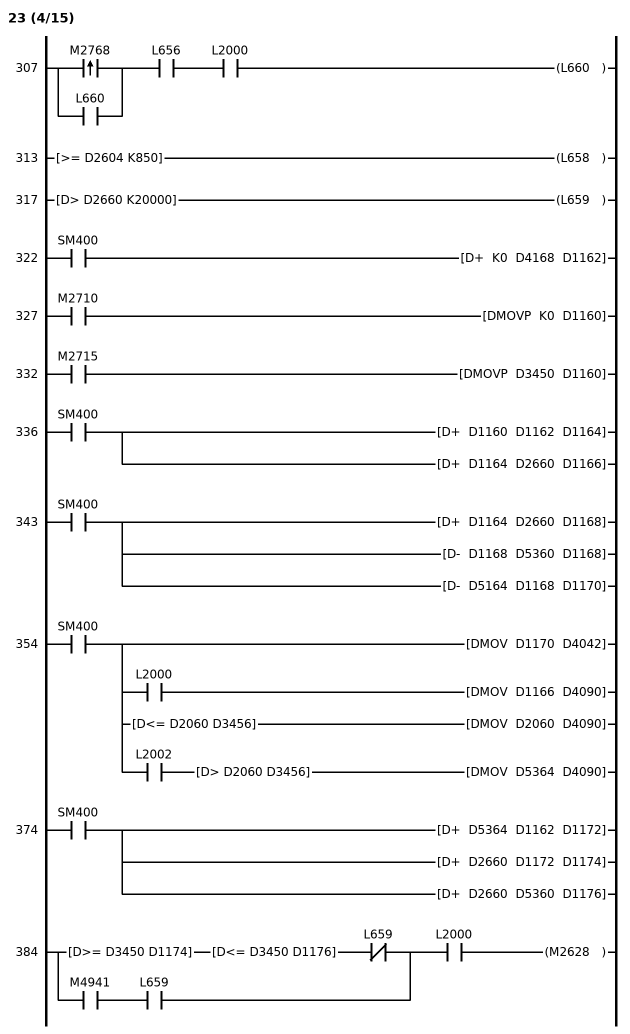
307   LDP     M2768
      OR      L660
      AND     L656
      AND     L2000
      OUT     L660
313   LD>=    D2604 K850
      OUT     L658
317   LDD>    D2660 K20000
      OUT     L659
322   LD      SM400
      D+      K0 D4168 D1162
327   LD      M2710
      DMOVP   K0 D1160
332   LD      M2715
      DMOVP   D3450 D1160
336   LD      SM400
      D+      D1160 D1162 D1164
      D+      D1164 D2660 D1166
343   LD      SM400
      D+      D1164 D2660 D1168
      D-      D1168 D5360 D1168
      D-      D5164 D1168 D1170
354   LD      SM400
      DMOV    D1170 D4042
      MPS
      AND     L2000
      DMOV    D1166 D4090
      MRD
      ANDD<=  D2060 D3456
      DMOV    D2060 D4090
      MPP
      AND     L2002
      ANDD>   D2060 D3456
      DMOV    D5364 D4090
374   LD      SM400
      D+      D5364 D1162 D1172
      D+      D2660 D1172 D1174
      D+      D2660 D5360 D1176
384   LDD>=   D3450 D1174
      ANDD<=  D3450 D1176
      ANI     L659
      LD      M4941
      AND     L659
      ORB
      AND     L2000
      OUT     M2628
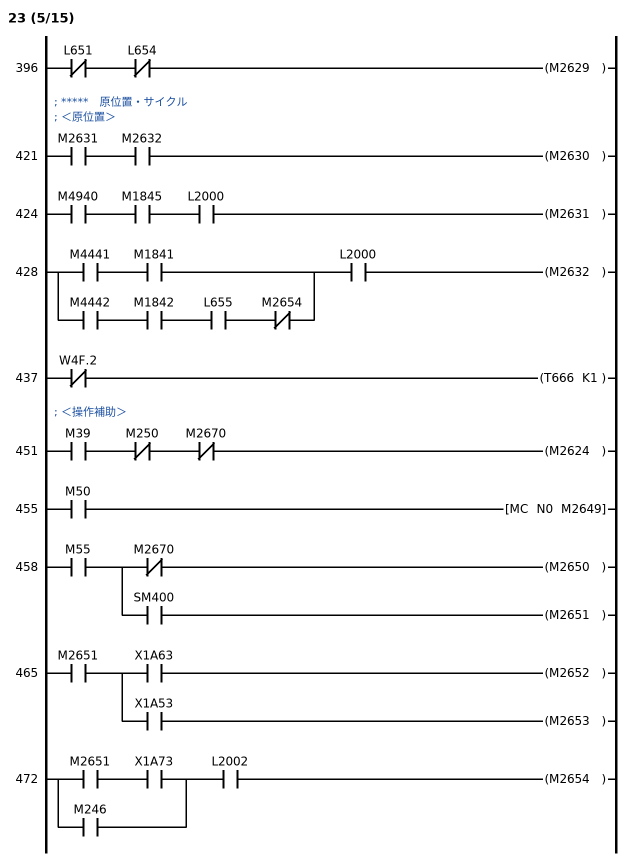
396   LDI     L651
      ANI     L654
      OUT     M2629
; *****　原位置・サイクル
; ＜原位置＞
421   LD      M2631
      AND     M2632
      OUT     M2630
424   LD      M4940
      AND     M1845
      AND     L2000
      OUT     M2631
428   LD      M4441
      AND     M1841
      LD      M4442
      AND     M1842
      AND     L655
      ANI     M2654
      ORB
      AND     L2000
      OUT     M2632
437   LDI     W4F.2
      OUT     T666 K1
; ＜操作補助＞
451   LD      M39
      ANI     M250
      ANI     M2670
      OUT     M2624
455   LD      M50
      MC      N0 M2649
458   LD      M55
      MPS
      ANI     M2670
      OUT     M2650
      MPP
      AND     SM400
      OUT     M2651
465   LD      M2651
      MPS
      AND     X1A63
      OUT     M2652
      MPP
      AND     X1A53
      OUT     M2653
472   LD      M2651
      AND     X1A73
      OR      M246
      AND     L2002
      OUT     M2654
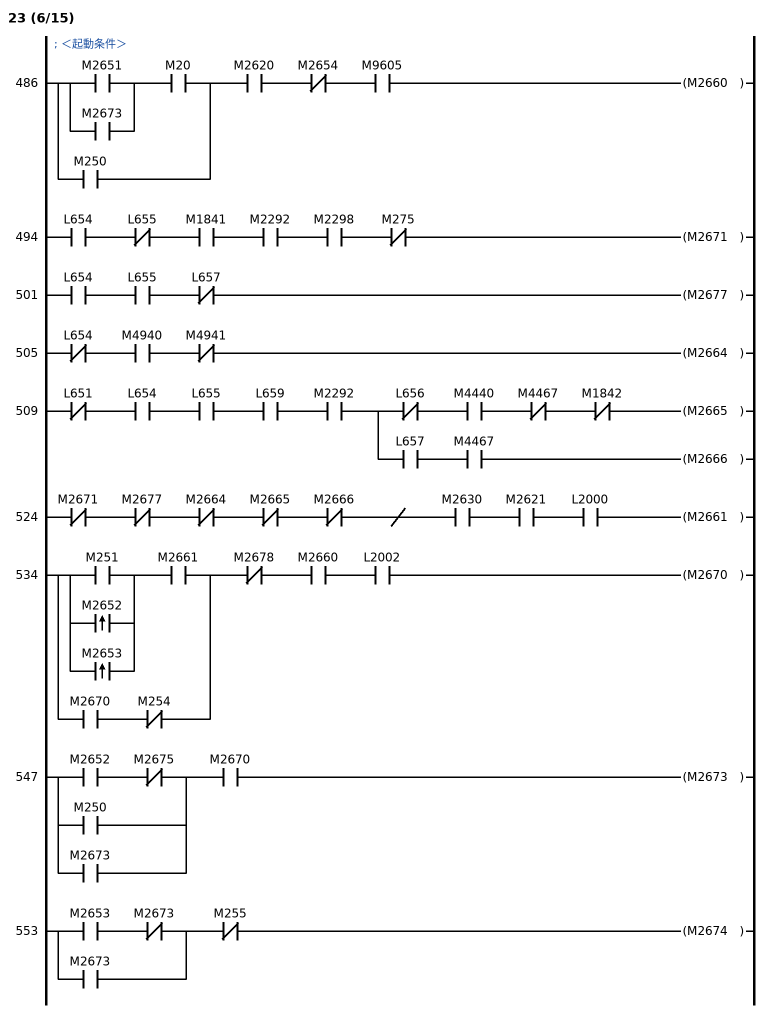
; ＜起動条件＞
486   LD      M2651
      OR      M2673
      AND     M20
      OR      M250
      AND     M2620
      ANI     M2654
      AND     M9605
      OUT     M2660
494   LD      L654
      ANI     L655
      AND     M1841
      AND     M2292
      AND     M2298
      ANI     M275
      OUT     M2671
501   LD      L654
      AND     L655
      ANI     L657
      OUT     M2677
505   LDI     L654
      AND     M4940
      ANI     M4941
      OUT     M2664
509   LDI     L651
      AND     L654
      AND     L655
      AND     L659
      AND     M2292
      MPS
      ANI     L656
      AND     M4440
      ANI     M4467
      ANI     M1842
      OUT     M2665
      MPP
      AND     L657
      AND     M4467
      OUT     M2666
524   LDI     M2671
      ANI     M2677
      ANI     M2664
      ANI     M2665
      ANI     M2666
      INV
      AND     M2630
      AND     M2621
      AND     L2000
      OUT     M2661
534   LD      M251
      ORP     M2652
      ORP     M2653
      AND     M2661
      LD      M2670
      ANI     M254
      ORB
      ANI     M2678
      AND     M2660
      AND     L2002
      OUT     M2670
547   LD      M2652
      ANI     M2675
      OR      M250
      OR      M2673
      AND     M2670
      OUT     M2673
553   LD      M2653
      ANI     M2673
      OR      M2673
      ANI     M255
      OUT     M2674
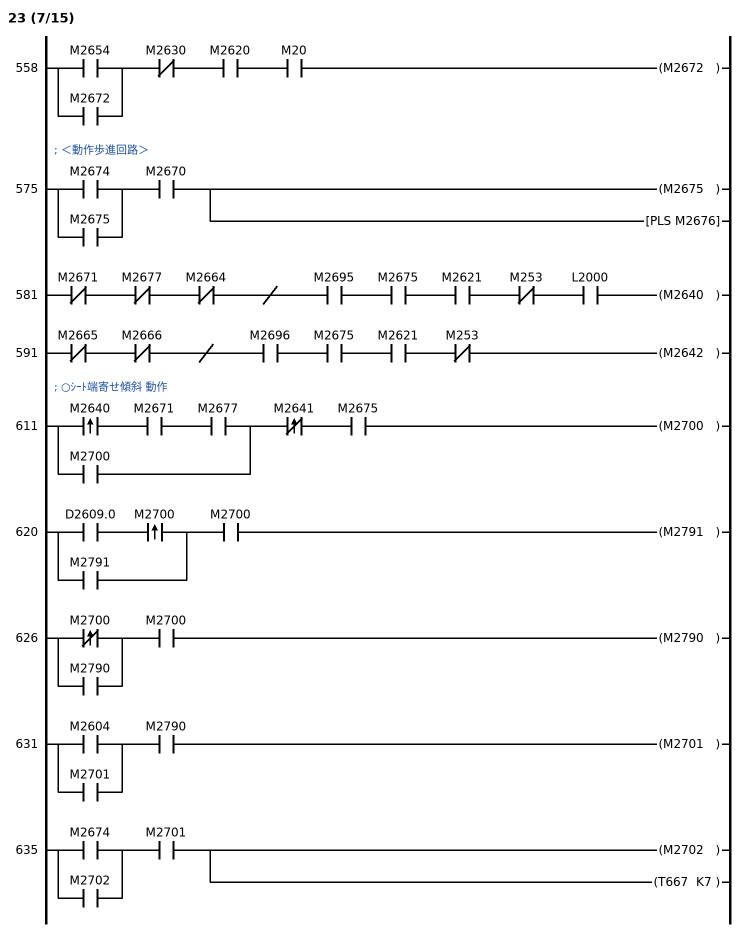
558   LD      M2654
      OR      M2672
      ANI     M2630
      AND     M2620
      AND     M20
      OUT     M2672
; ＜動作歩進回路＞
575   LD      M2674
      OR      M2675
      AND     M2670
      OUT     M2675
      PLS     M2676
581   LDI     M2671
      ANI     M2677
      ANI     M2664
      INV
      AND     M2695
      AND     M2675
      AND     M2621
      ANI     M253
      AND     L2000
      OUT     M2640
591   LDI     M2665
      ANI     M2666
      INV
      AND     M2696
      AND     M2675
      AND     M2621
      ANI     M253
      OUT     M2642
; ○ｼｰﾄ端寄せ傾斜 動作
611   LDP     M2640
      AND     M2671
      AND     M2677
      OR      M2700
      ANDPI   M2641
      AND     M2675
      OUT     M2700
620   LD      D2609.0
      ANDP    M2700
      OR      M2791
      AND     M2700
      OUT     M2791
626   LDPI    M2700
      OR      M2790
      AND     M2700
      OUT     M2790
631   LD      M2604
      OR      M2701
      AND     M2790
      OUT     M2701
635   LD      M2674
      OR      M2702
      AND     M2701
      OUT     M2702
      OUT     T667 K7
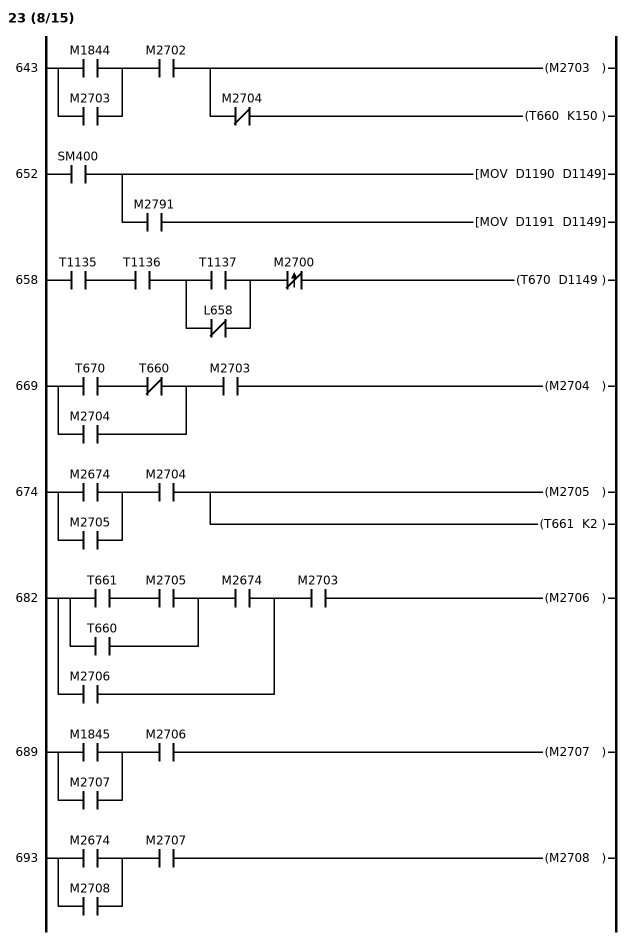
643   LD      M1844
      OR      M2703
      AND     M2702
      OUT     M2703
      ANI     M2704
      OUT     T660 K150
652   LD      SM400
      MOV     D1190 D1149
      AND     M2791
      MOV     D1191 D1149
658   LD      T1135
      AND     T1136
      LD      T1137
      ORI     L658
      ANB
      ANDPI   M2700
      OUT     T670 D1149
669   LD      T670
      ANI     T660
      OR      M2704
      AND     M2703
      OUT     M2704
674   LD      M2674
      OR      M2705
      AND     M2704
      OUT     M2705
      OUT     T661 K2
682   LD      T661
      AND     M2705
      OR      T660
      AND     M2674
      OR      M2706
      AND     M2703
      OUT     M2706
689   LD      M1845
      OR      M2707
      AND     M2706
      OUT     M2707
693   LD      M2674
      OR      M2708
      AND     M2707
      OUT     M2708
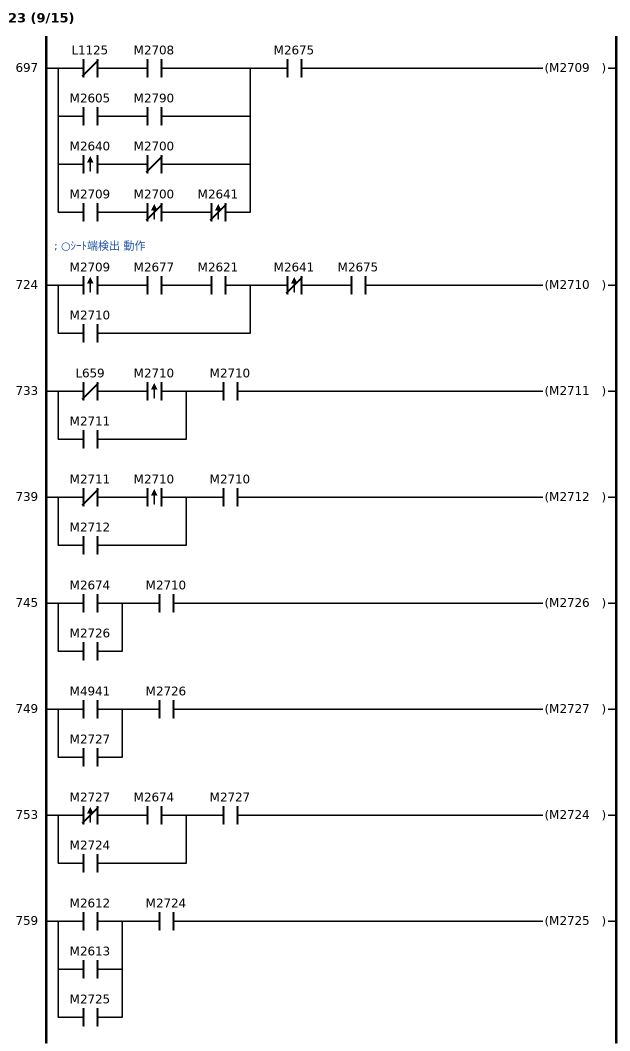
697   LDI     L1125
      AND     M2708
      LD      M2605
      AND     M2790
      ORB
      LDP     M2640
      ANI     M2700
      ORB
      LD      M2709
      ANDPI   M2700
      ANDPI   M2641
      ORB
      AND     M2675
      OUT     M2709
; ○ｼｰﾄ端検出 動作
724   LDP     M2709
      AND     M2677
      AND     M2621
      OR      M2710
      ANDPI   M2641
      AND     M2675
      OUT     M2710
733   LDI     L659
      ANDP    M2710
      OR      M2711
      AND     M2710
      OUT     M2711
739   LDI     M2711
      ANDP    M2710
      OR      M2712
      AND     M2710
      OUT     M2712
745   LD      M2674
      OR      M2726
      AND     M2710
      OUT     M2726
749   LD      M4941
      OR      M2727
      AND     M2726
      OUT     M2727
753   LDPI    M2727
      AND     M2674
      OR      M2724
      AND     M2727
      OUT     M2724
759   LD      M2612
      OR      M2613
      OR      M2725
      AND     M2724
      OUT     M2725
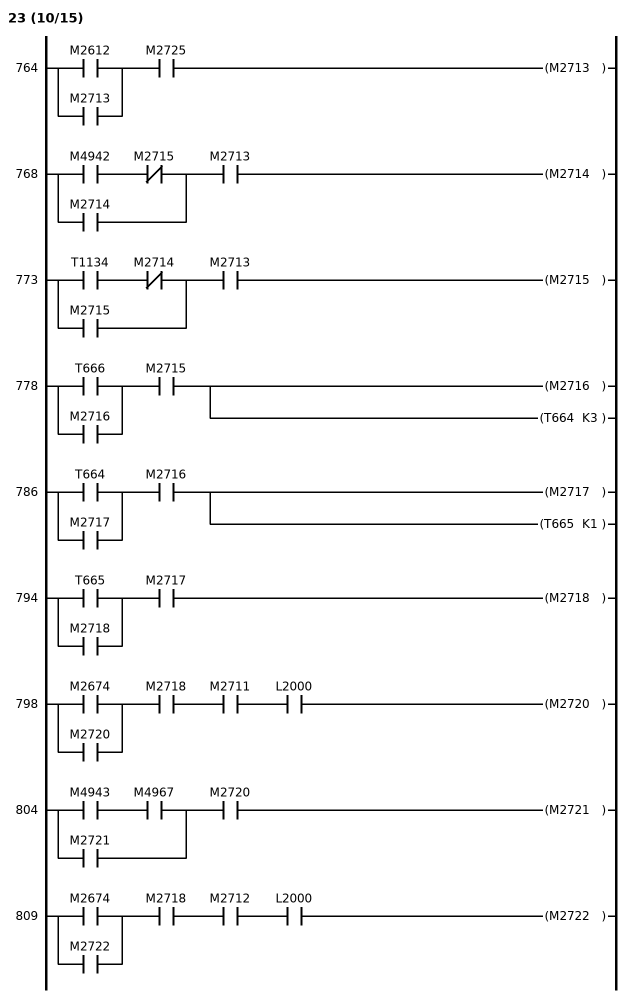
764   LD      M2612
      OR      M2713
      AND     M2725
      OUT     M2713
768   LD      M4942
      ANI     M2715
      OR      M2714
      AND     M2713
      OUT     M2714
773   LD      T1134
      ANI     M2714
      OR      M2715
      AND     M2713
      OUT     M2715
778   LD      T666
      OR      M2716
      AND     M2715
      OUT     M2716
      OUT     T664 K3
786   LD      T664
      OR      M2717
      AND     M2716
      OUT     M2717
      OUT     T665 K1
794   LD      T665
      OR      M2718
      AND     M2717
      OUT     M2718
798   LD      M2674
      OR      M2720
      AND     M2718
      AND     M2711
      AND     L2000
      OUT     M2720
804   LD      M4943
      AND     M4967
      OR      M2721
      AND     M2720
      OUT     M2721
809   LD      M2674
      OR      M2722
      AND     M2718
      AND     M2712
      AND     L2000
      OUT     M2722
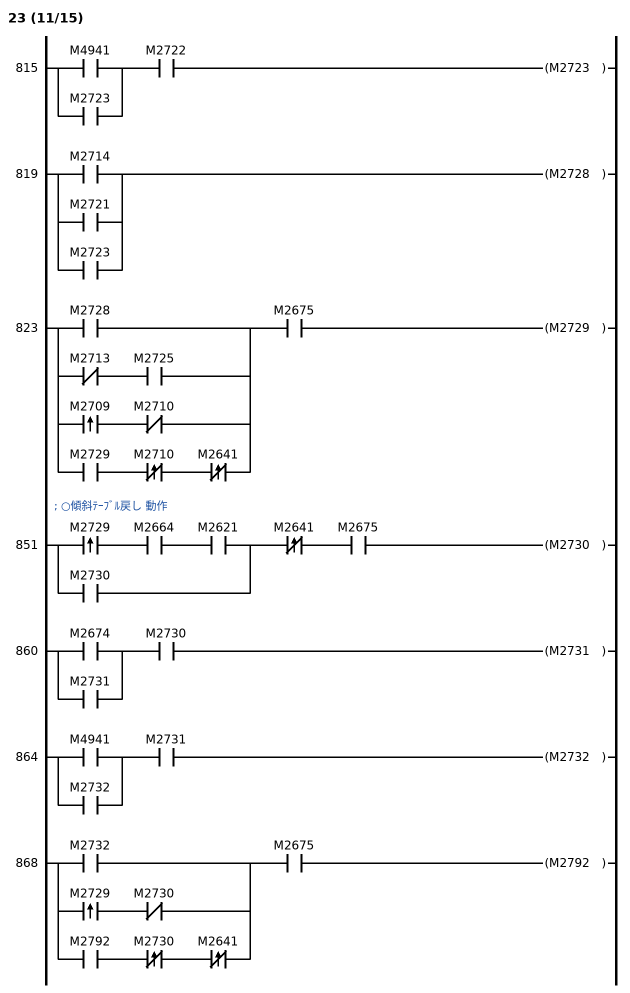
815   LD      M4941
      OR      M2723
      AND     M2722
      OUT     M2723
819   LD      M2714
      OR      M2721
      OR      M2723
      OUT     M2728
823   LD      M2728
      LDI     M2713
      AND     M2725
      ORB
      LDP     M2709
      ANI     M2710
      ORB
      LD      M2729
      ANDPI   M2710
      ANDPI   M2641
      ORB
      AND     M2675
      OUT     M2729
; ○傾斜ﾃｰﾌﾞﾙ戻し 動作
851   LDP     M2729
      AND     M2664
      AND     M2621
      OR      M2730
      ANDPI   M2641
      AND     M2675
      OUT     M2730
860   LD      M2674
      OR      M2731
      AND     M2730
      OUT     M2731
864   LD      M4941
      OR      M2732
      AND     M2731
      OUT     M2732
868   LD      M2732
      LDP     M2729
      ANI     M2730
      ORB
      LD      M2792
      ANDPI   M2730
      ANDPI   M2641
      ORB
      AND     M2675
      OUT     M2792
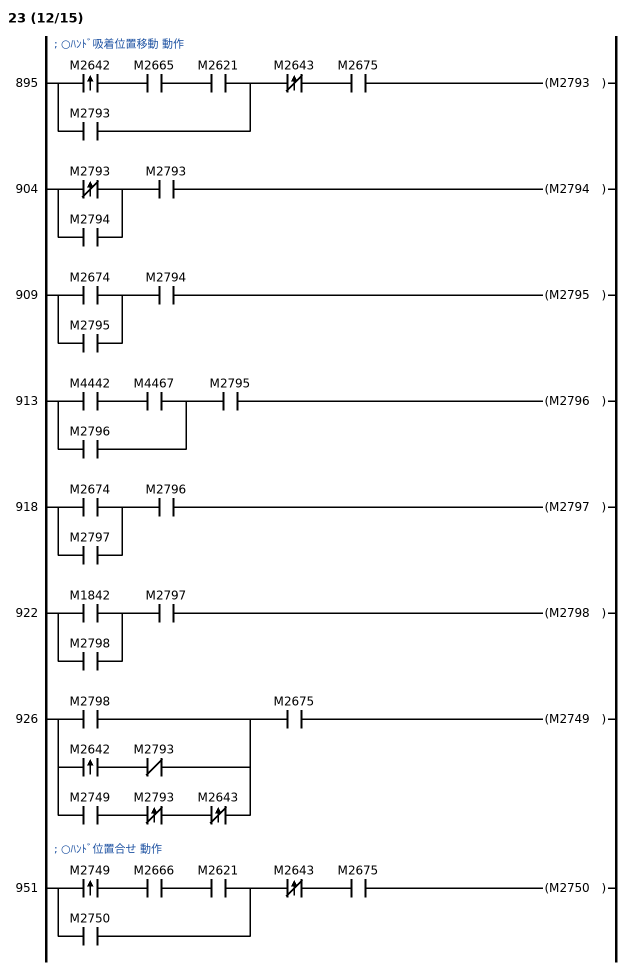
; ○ﾊﾝﾄﾞ吸着位置移動 動作
895   LDP     M2642
      AND     M2665
      AND     M2621
      OR      M2793
      ANDPI   M2643
      AND     M2675
      OUT     M2793
904   LDPI    M2793
      OR      M2794
      AND     M2793
      OUT     M2794
909   LD      M2674
      OR      M2795
      AND     M2794
      OUT     M2795
913   LD      M4442
      AND     M4467
      OR      M2796
      AND     M2795
      OUT     M2796
918   LD      M2674
      OR      M2797
      AND     M2796
      OUT     M2797
922   LD      M1842
      OR      M2798
      AND     M2797
      OUT     M2798
926   LD      M2798
      LDP     M2642
      ANI     M2793
      ORB
      LD      M2749
      ANDPI   M2793
      ANDPI   M2643
      ORB
      AND     M2675
      OUT     M2749
; ○ﾊﾝﾄﾞ位置合せ 動作
951   LDP     M2749
      AND     M2666
      AND     M2621
      OR      M2750
      ANDPI   M2643
      AND     M2675
      OUT     M2750
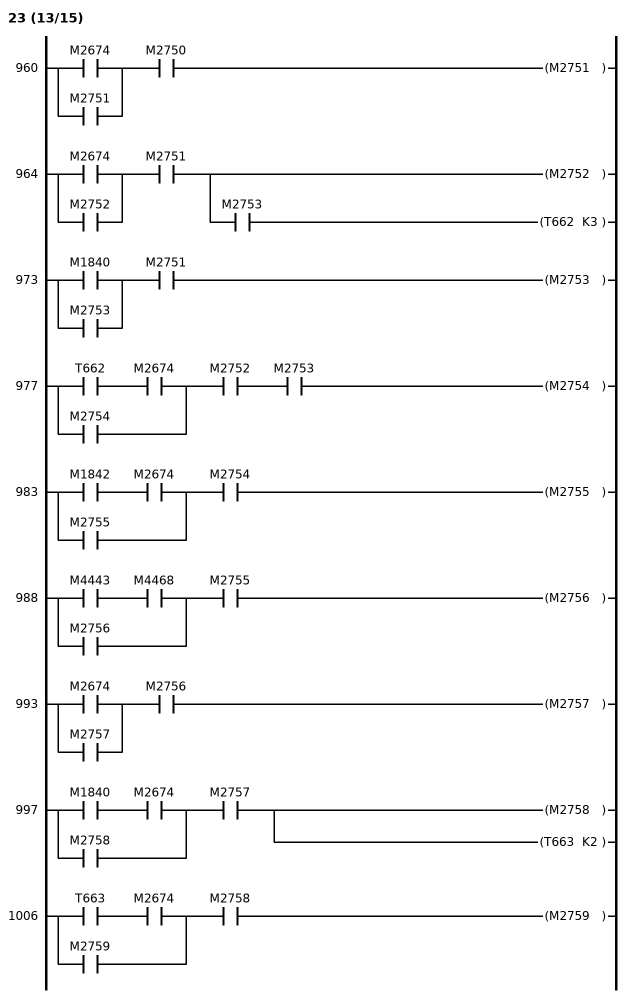
960   LD      M2674
      OR      M2751
      AND     M2750
      OUT     M2751
964   LD      M2674
      OR      M2752
      AND     M2751
      OUT     M2752
      AND     M2753
      OUT     T662 K3
973   LD      M1840
      OR      M2753
      AND     M2751
      OUT     M2753
977   LD      T662
      AND     M2674
      OR      M2754
      AND     M2752
      AND     M2753
      OUT     M2754
983   LD      M1842
      AND     M2674
      OR      M2755
      AND     M2754
      OUT     M2755
988   LD      M4443
      AND     M4468
      OR      M2756
      AND     M2755
      OUT     M2756
993   LD      M2674
      OR      M2757
      AND     M2756
      OUT     M2757
997   LD      M1840
      AND     M2674
      OR      M2758
      AND     M2757
      OUT     M2758
      OUT     T663 K2
1006  LD      T663
      AND     M2674
      OR      M2759
      AND     M2758
      OUT     M2759
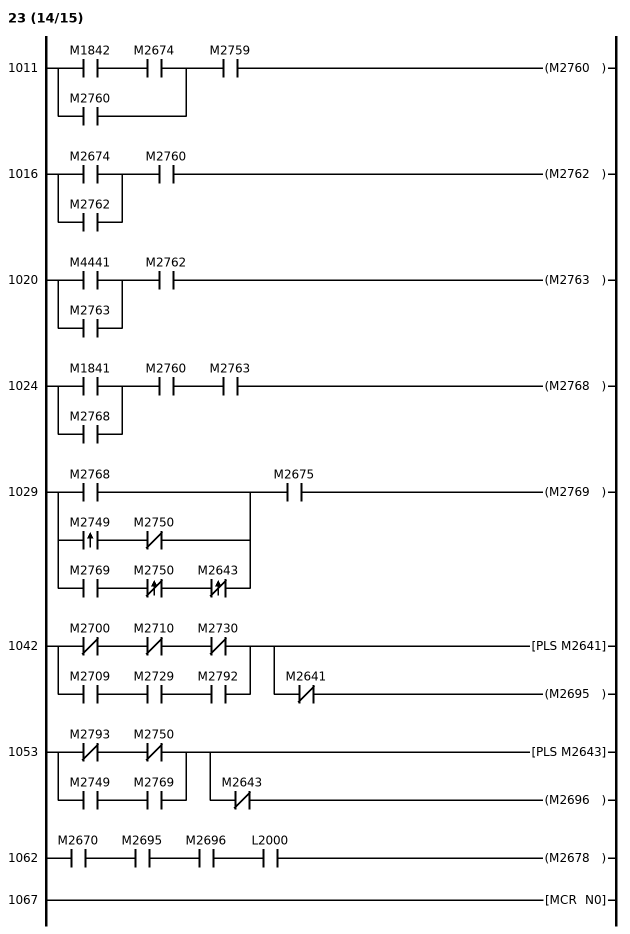
1011  LD      M1842
      AND     M2674
      OR      M2760
      AND     M2759
      OUT     M2760
1016  LD      M2674
      OR      M2762
      AND     M2760
      OUT     M2762
1020  LD      M4441
      OR      M2763
      AND     M2762
      OUT     M2763
1024  LD      M1841
      OR      M2768
      AND     M2760
      AND     M2763
      OUT     M2768
1029  LD      M2768
      LDP     M2749
      ANI     M2750
      ORB
      LD      M2769
      ANDPI   M2750
      ANDPI   M2643
      ORB
      AND     M2675
      OUT     M2769
1042  LDI     M2700
      ANI     M2710
      ANI     M2730
      LD      M2709
      AND     M2729
      AND     M2792
      ORB
      PLS     M2641
      ANI     M2641
      OUT     M2695
1053  LDI     M2793
      ANI     M2750
      LD      M2749
      AND     M2769
      ORB
      PLS     M2643
      ANI     M2643
      OUT     M2696
1062  LD      M2670
      AND     M2695
      AND     M2696
      AND     L2000
      OUT     M2678
1067  MCR     N0
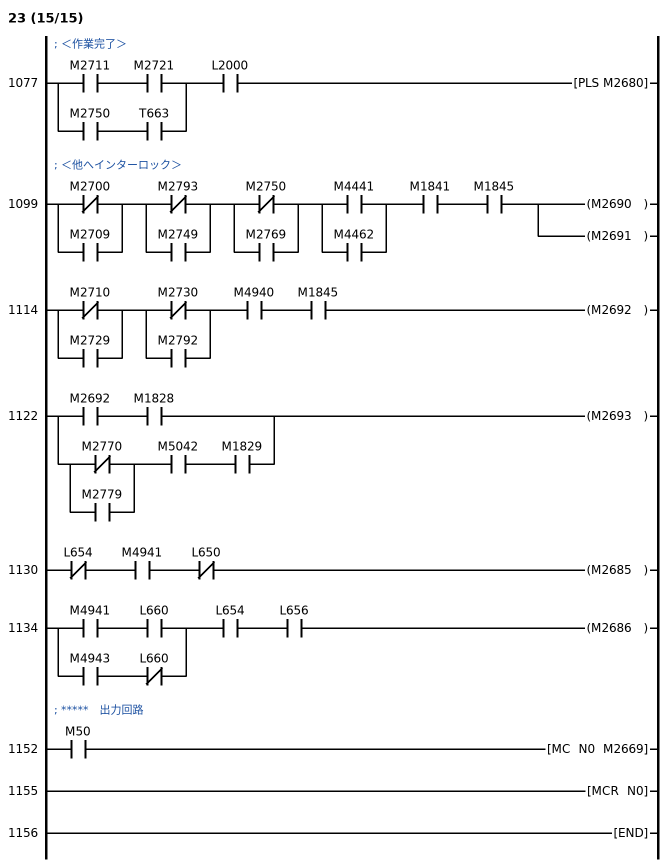
; ＜作業完了＞
1077  LD      M2711
      AND     M2721
      LD      M2750
      AND     T663
      ORB
      AND     L2000
      PLS     M2680
; ＜他へインターロック＞
1099  LDI     M2700
      OR      M2709
      LDI     M2793
      OR      M2749
      ANB
      LDI     M2750
      OR      M2769
      ANB
      LD      M4441
      OR      M4462
      ANB
      AND     M1841
      AND     M1845
      OUT     M2690
      OUT     M2691
1114  LDI     M2710
      OR      M2729
      LDI     M2730
      OR      M2792
      ANB
      AND     M4940
      AND     M1845
      OUT     M2692
1122  LD      M2692
      AND     M1828
      LDI     M2770
      OR      M2779
      AND     M5042
      AND     M1829
      ORB
      OUT     M2693
1130  LDI     L654
      AND     M4941
      ANI     L650
      OUT     M2685
1134  LD      M4941
      AND     L660
      LD      M4943
      ANI     L660
      ORB
      AND     L654
      AND     L656
      OUT     M2686
; *****　出力回路
1152  LD      M50
      MC      N0 M2669
1155  MCR     N0
1156  END
END_PROGRAM

PROGRAM 24
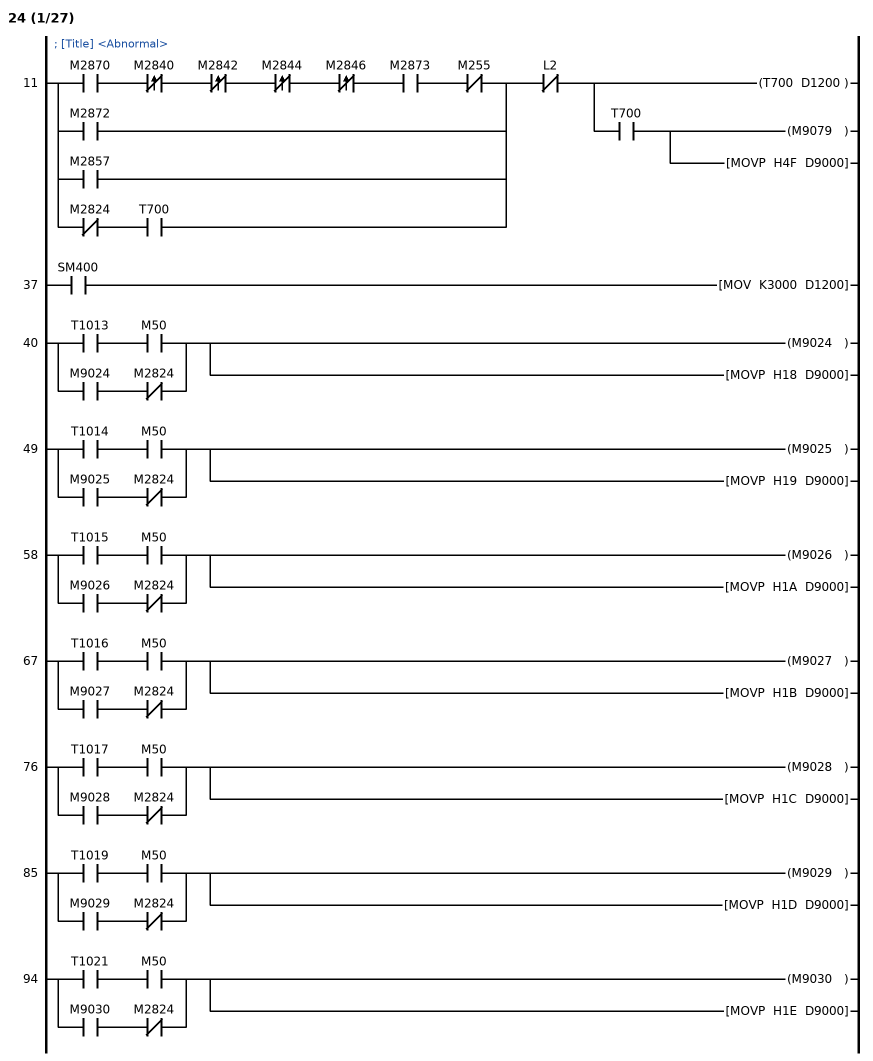
; [Title] <Abnormal>
11    LD      M2870
      ANDPI   M2840
      ANDPI   M2842
      ANDPI   M2844
      ANDPI   M2846
      AND     M2873
      ANI     M255
      OR      M2872
      OR      M2857
      LDI     M2824
      AND     T700
      ORB
      ANI     L2
      OUT     T700 D1200
      AND     T700
      OUT     M9079
      MOVP    H4F D9000
37    LD      SM400
      MOV     K3000 D1200
40    LD      T1013
      AND     M50
      LD      M9024
      ANI     M2824
      ORB
      OUT     M9024
      MOVP    H18 D9000
49    LD      T1014
      AND     M50
      LD      M9025
      ANI     M2824
      ORB
      OUT     M9025
      MOVP    H19 D9000
58    LD      T1015
      AND     M50
      LD      M9026
      ANI     M2824
      ORB
      OUT     M9026
      MOVP    H1A D9000
67    LD      T1016
      AND     M50
      LD      M9027
      ANI     M2824
      ORB
      OUT     M9027
      MOVP    H1B D9000
76    LD      T1017
      AND     M50
      LD      M9028
      ANI     M2824
      ORB
      OUT     M9028
      MOVP    H1C D9000
85    LD      T1019
      AND     M50
      LD      M9029
      ANI     M2824
      ORB
      OUT     M9029
      MOVP    H1D D9000
94    LD      T1021
      AND     M50
      LD      M9030
      ANI     M2824
      ORB
      OUT     M9030
      MOVP    H1E D9000
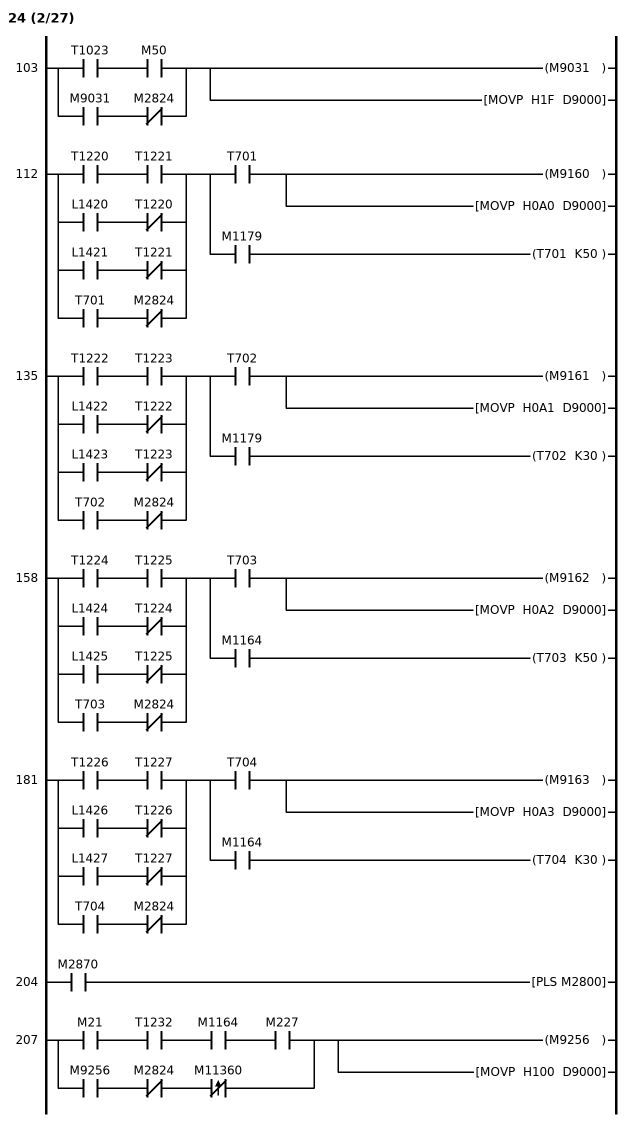
103   LD      T1023
      AND     M50
      LD      M9031
      ANI     M2824
      ORB
      OUT     M9031
      MOVP    H1F D9000
112   LD      T1220
      AND     T1221
      LD      L1420
      ANI     T1220
      ORB
      LD      L1421
      ANI     T1221
      ORB
      LD      T701
      ANI     M2824
      ORB
      MPS
      AND     T701
      OUT     M9160
      MOVP    H0A0 D9000
      MPP
      AND     M1179
      OUT     T701 K50
135   LD      T1222
      AND     T1223
      LD      L1422
      ANI     T1222
      ORB
      LD      L1423
      ANI     T1223
      ORB
      LD      T702
      ANI     M2824
      ORB
      MPS
      AND     T702
      OUT     M9161
      MOVP    H0A1 D9000
      MPP
      AND     M1179
      OUT     T702 K30
158   LD      T1224
      AND     T1225
      LD      L1424
      ANI     T1224
      ORB
      LD      L1425
      ANI     T1225
      ORB
      LD      T703
      ANI     M2824
      ORB
      MPS
      AND     T703
      OUT     M9162
      MOVP    H0A2 D9000
      MPP
      AND     M1164
      OUT     T703 K50
181   LD      T1226
      AND     T1227
      LD      L1426
      ANI     T1226
      ORB
      LD      L1427
      ANI     T1227
      ORB
      LD      T704
      ANI     M2824
      ORB
      MPS
      AND     T704
      OUT     M9163
      MOVP    H0A3 D9000
      MPP
      AND     M1164
      OUT     T704 K30
204   LD      M2870
      PLS     M2800
207   LD      M21
      AND     T1232
      AND     M1164
      AND     M227
      LD      M9256
      ANI     M2824
      ANDPI   M11360
      ORB
      OUT     M9256
      MOVP    H100 D9000
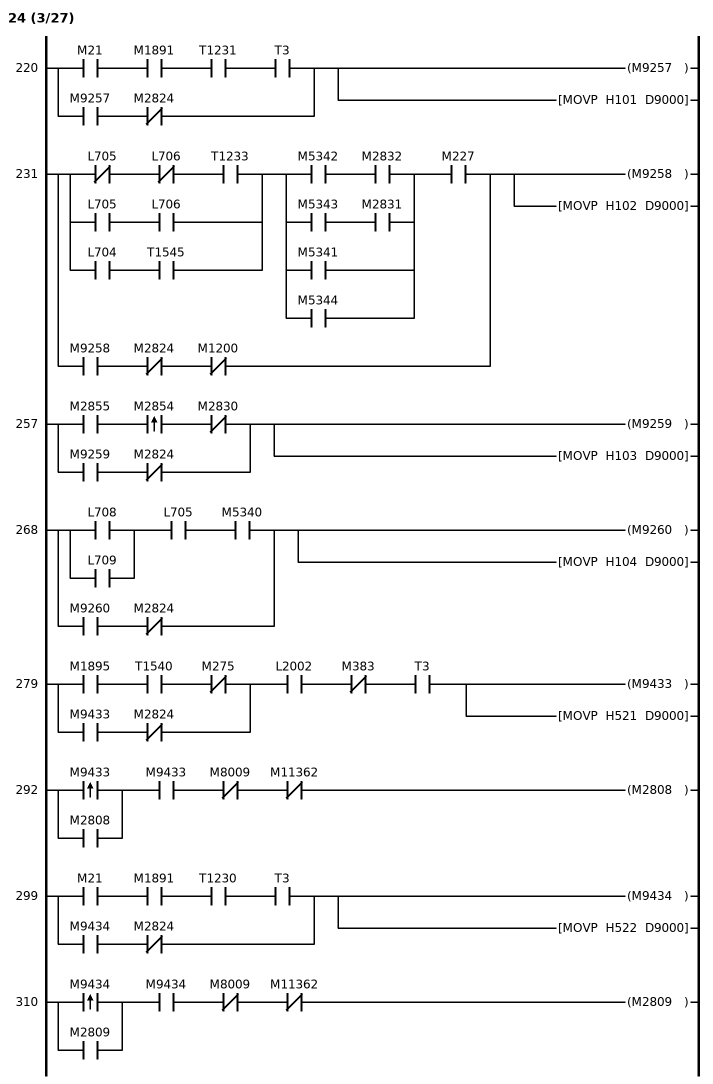
220   LD      M21
      AND     M1891
      AND     T1231
      AND     T3
      LD      M9257
      ANI     M2824
      ORB
      OUT     M9257
      MOVP    H101 D9000
231   LDI     L705
      ANI     L706
      AND     T1233
      LD      L705
      AND     L706
      ORB
      LD      L704
      AND     T1545
      ORB
      LD      M5342
      AND     M2832
      LD      M5343
      AND     M2831
      ORB
      OR      M5341
      OR      M5344
      ANB
      AND     M227
      LD      M9258
      ANI     M2824
      ANI     M1200
      ORB
      OUT     M9258
      MOVP    H102 D9000
257   LD      M2855
      ANDP    M2854
      ANI     M2830
      LD      M9259
      ANI     M2824
      ORB
      OUT     M9259
      MOVP    H103 D9000
268   LD      L708
      OR      L709
      AND     L705
      AND     M5340
      LD      M9260
      ANI     M2824
      ORB
      OUT     M9260
      MOVP    H104 D9000
279   LD      M1895
      AND     T1540
      ANI     M275
      LD      M9433
      ANI     M2824
      ORB
      AND     L2002
      ANI     M383
      AND     T3
      OUT     M9433
      MOVP    H521 D9000
292   LDP     M9433
      OR      M2808
      AND     M9433
      ANI     M8009
      ANI     M11362
      OUT     M2808
299   LD      M21
      AND     M1891
      AND     T1230
      AND     T3
      LD      M9434
      ANI     M2824
      ORB
      OUT     M9434
      MOVP    H522 D9000
310   LDP     M9434
      OR      M2809
      AND     M9434
      ANI     M8009
      ANI     M11362
      OUT     M2809
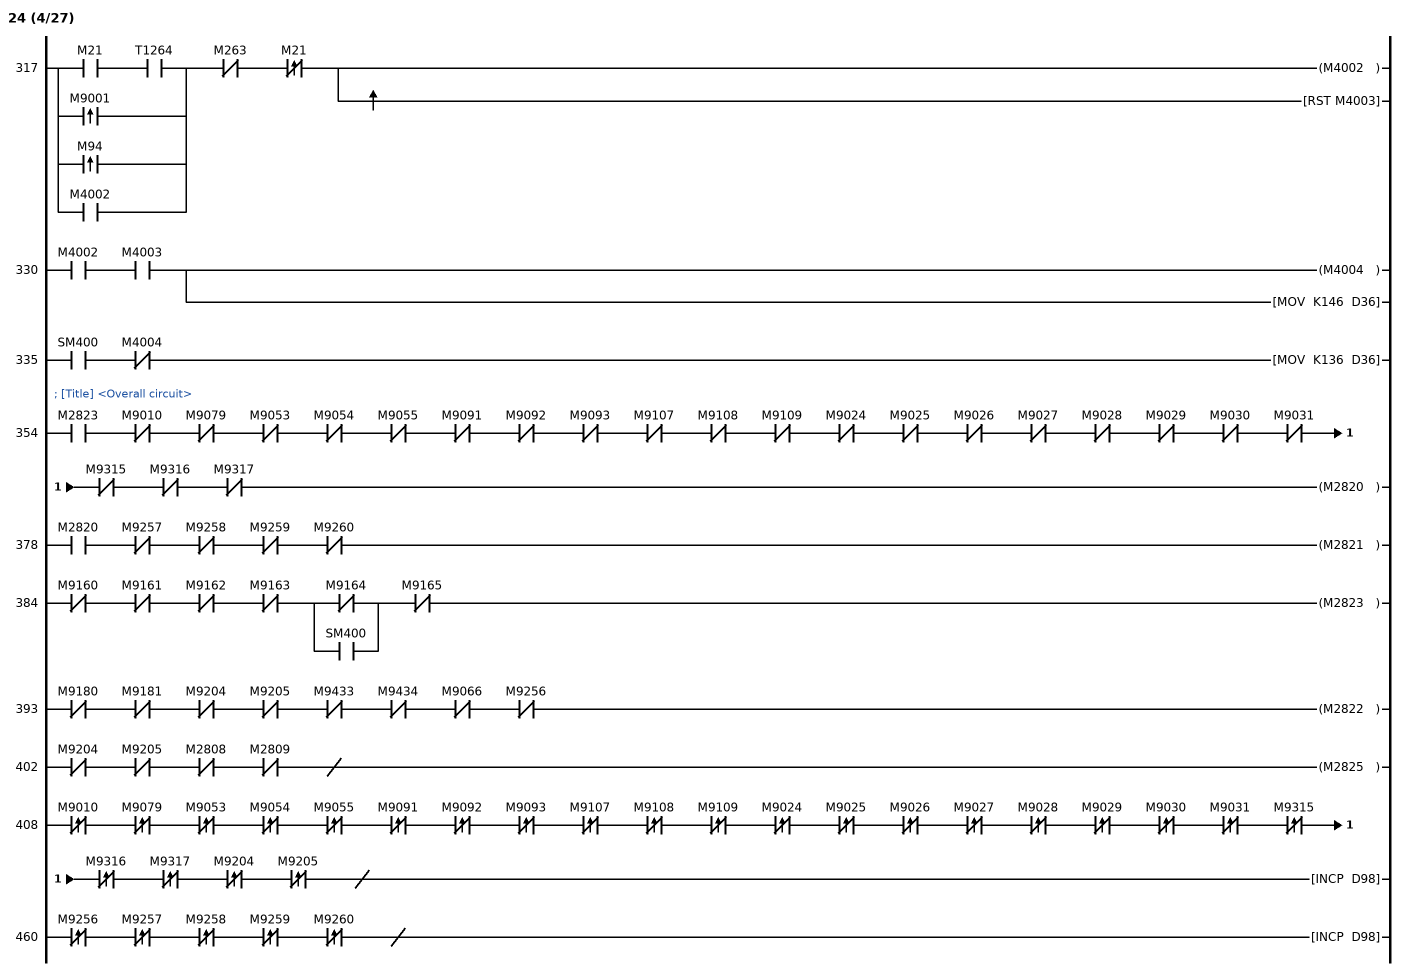
317   LD      M21
      AND     T1264
      ORP     M9001
      ORP     M94
      OR      M4002
      ANI     M263
      ANDPI   M21
      OUT     M4002
      MEP
      RST     M4003
330   LD      M4002
      AND     M4003
      OUT     M4004
      MOV     K146 D36
335   LD      SM400
      ANI     M4004
      MOV     K136 D36
; [Title] <Overall circuit>
354   LD      M2823
      ANI     M9010
      ANI     M9079
      ANI     M9053
      ANI     M9054
      ANI     M9055
      ANI     M9091
      ANI     M9092
      ANI     M9093
      ANI     M9107
      ANI     M9108
      ANI     M9109
      ANI     M9024
      ANI     M9025
      ANI     M9026
      ANI     M9027
      ANI     M9028
      ANI     M9029
      ANI     M9030
      ANI     M9031
      ANI     M9315
      ANI     M9316
      ANI     M9317
      OUT     M2820
378   LD      M2820
      ANI     M9257
      ANI     M9258
      ANI     M9259
      ANI     M9260
      OUT     M2821
384   LDI     M9160
      ANI     M9161
      ANI     M9162
      ANI     M9163
      LDI     M9164
      OR      SM400
      ANB
      ANI     M9165
      OUT     M2823
393   LDI     M9180
      ANI     M9181
      ANI     M9204
      ANI     M9205
      ANI     M9433
      ANI     M9434
      ANI     M9066
      ANI     M9256
      OUT     M2822
402   LDI     M9204
      ANI     M9205
      ANI     M2808
      ANI     M2809
      INV
      OUT     M2825
408   LDPI    M9010
      ANDPI   M9079
      ANDPI   M9053
      ANDPI   M9054
      ANDPI   M9055
      ANDPI   M9091
      ANDPI   M9092
      ANDPI   M9093
      ANDPI   M9107
      ANDPI   M9108
      ANDPI   M9109
      ANDPI   M9024
      ANDPI   M9025
      ANDPI   M9026
      ANDPI   M9027
      ANDPI   M9028
      ANDPI   M9029
      ANDPI   M9030
      ANDPI   M9031
      ANDPI   M9315
      ANDPI   M9316
      ANDPI   M9317
      ANDPI   M9204
      ANDPI   M9205
      INV
      INCP    D98
460   LDPI    M9256
      ANDPI   M9257
      ANDPI   M9258
      ANDPI   M9259
      ANDPI   M9260
      INV
      INCP    D98
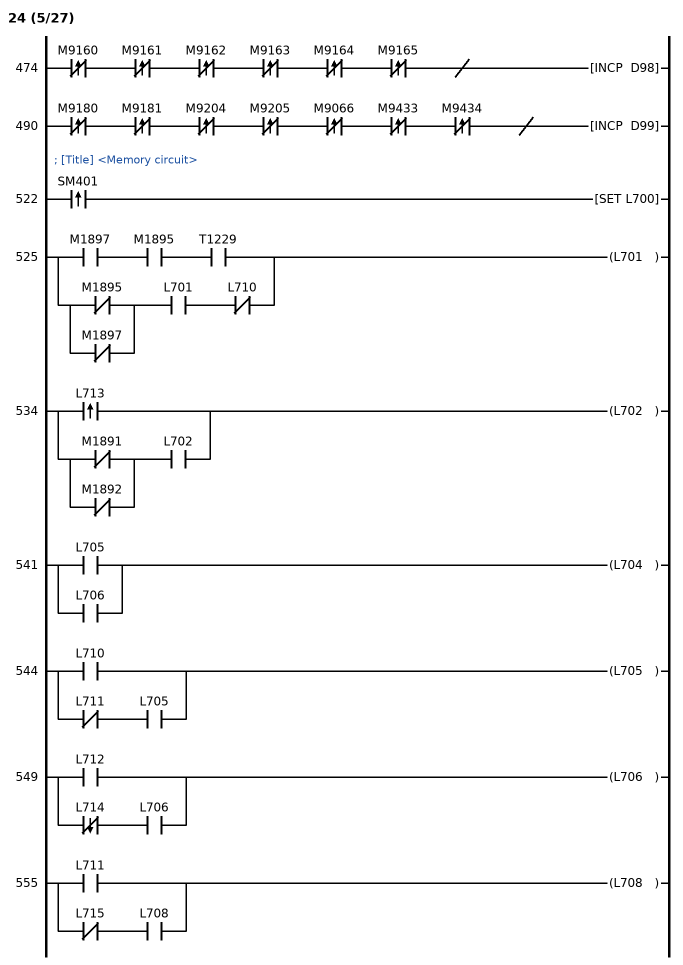
474   LDPI    M9160
      ANDPI   M9161
      ANDPI   M9162
      ANDPI   M9163
      ANDPI   M9164
      ANDPI   M9165
      INV
      INCP    D98
490   LDPI    M9180
      ANDPI   M9181
      ANDPI   M9204
      ANDPI   M9205
      ANDPI   M9066
      ANDPI   M9433
      ANDPI   M9434
      INV
      INCP    D99
; [Title] <Memory circuit>
522   LDP     SM401
      SET     L700
525   LD      M1897
      AND     M1895
      AND     T1229
      LDI     M1895
      ORI     M1897
      AND     L701
      ANI     L710
      ORB
      OUT     L701
534   LDP     L713
      LDI     M1891
      ORI     M1892
      AND     L702
      ORB
      OUT     L702
541   LD      L705
      OR      L706
      OUT     L704
544   LD      L710
      LDI     L711
      AND     L705
      ORB
      OUT     L705
549   LD      L712
      LDFI    L714
      AND     L706
      ORB
      OUT     L706
555   LD      L711
      LDI     L715
      AND     L708
      ORB
      OUT     L708
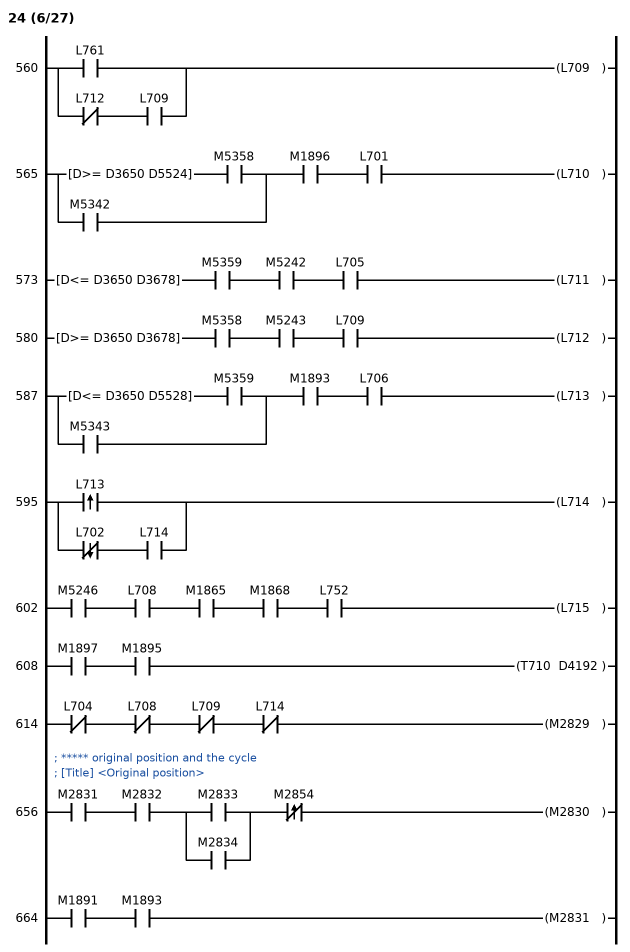
560   LD      L761
      LDI     L712
      AND     L709
      ORB
      OUT     L709
565   LDD>=   D3650 D5524
      AND     M5358
      OR      M5342
      AND     M1896
      AND     L701
      OUT     L710
573   LDD<=   D3650 D3678
      AND     M5359
      AND     M5242
      AND     L705
      OUT     L711
580   LDD>=   D3650 D3678
      AND     M5358
      AND     M5243
      AND     L709
      OUT     L712
587   LDD<=   D3650 D5528
      AND     M5359
      OR      M5343
      AND     M1893
      AND     L706
      OUT     L713
595   LDP     L713
      LDFI    L702
      AND     L714
      ORB
      OUT     L714
602   LD      M5246
      AND     L708
      AND     M1865
      AND     M1868
      AND     L752
      OUT     L715
608   LD      M1897
      AND     M1895
      OUT     T710 D4192
614   LDI     L704
      ANI     L708
      ANI     L709
      ANI     L714
      OUT     M2829
; ***** original position and the cycle
; [Title] <Original position>
656   LD      M2831
      AND     M2832
      LD      M2833
      OR      M2834
      ANB
      ANDPI   M2854
      OUT     M2830
664   LD      M1891
      AND     M1893
      OUT     M2831
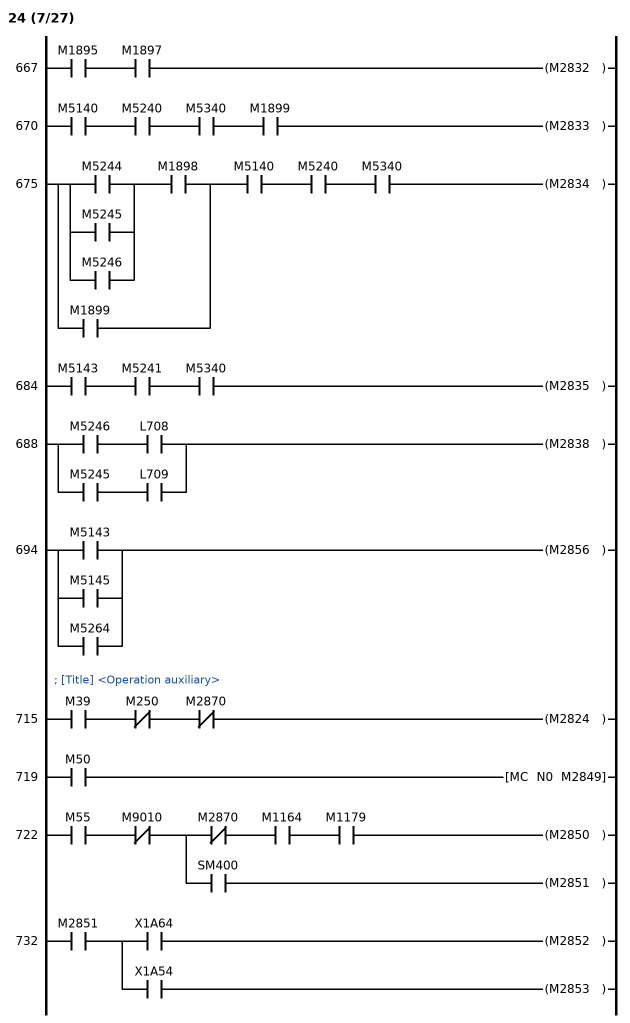
667   LD      M1895
      AND     M1897
      OUT     M2832
670   LD      M5140
      AND     M5240
      AND     M5340
      AND     M1899
      OUT     M2833
675   LD      M5244
      OR      M5245
      OR      M5246
      AND     M1898
      OR      M1899
      AND     M5140
      AND     M5240
      AND     M5340
      OUT     M2834
684   LD      M5143
      AND     M5241
      AND     M5340
      OUT     M2835
688   LD      M5246
      AND     L708
      LD      M5245
      AND     L709
      ORB
      OUT     M2838
694   LD      M5143
      OR      M5145
      OR      M5264
      OUT     M2856
; [Title] <Operation auxiliary>
715   LD      M39
      ANI     M250
      ANI     M2870
      OUT     M2824
719   LD      M50
      MC      N0 M2849
722   LD      M55
      ANI     M9010
      MPS
      ANI     M2870
      AND     M1164
      AND     M1179
      OUT     M2850
      MPP
      AND     SM400
      OUT     M2851
732   LD      M2851
      MPS
      AND     X1A64
      OUT     M2852
      MPP
      AND     X1A54
      OUT     M2853
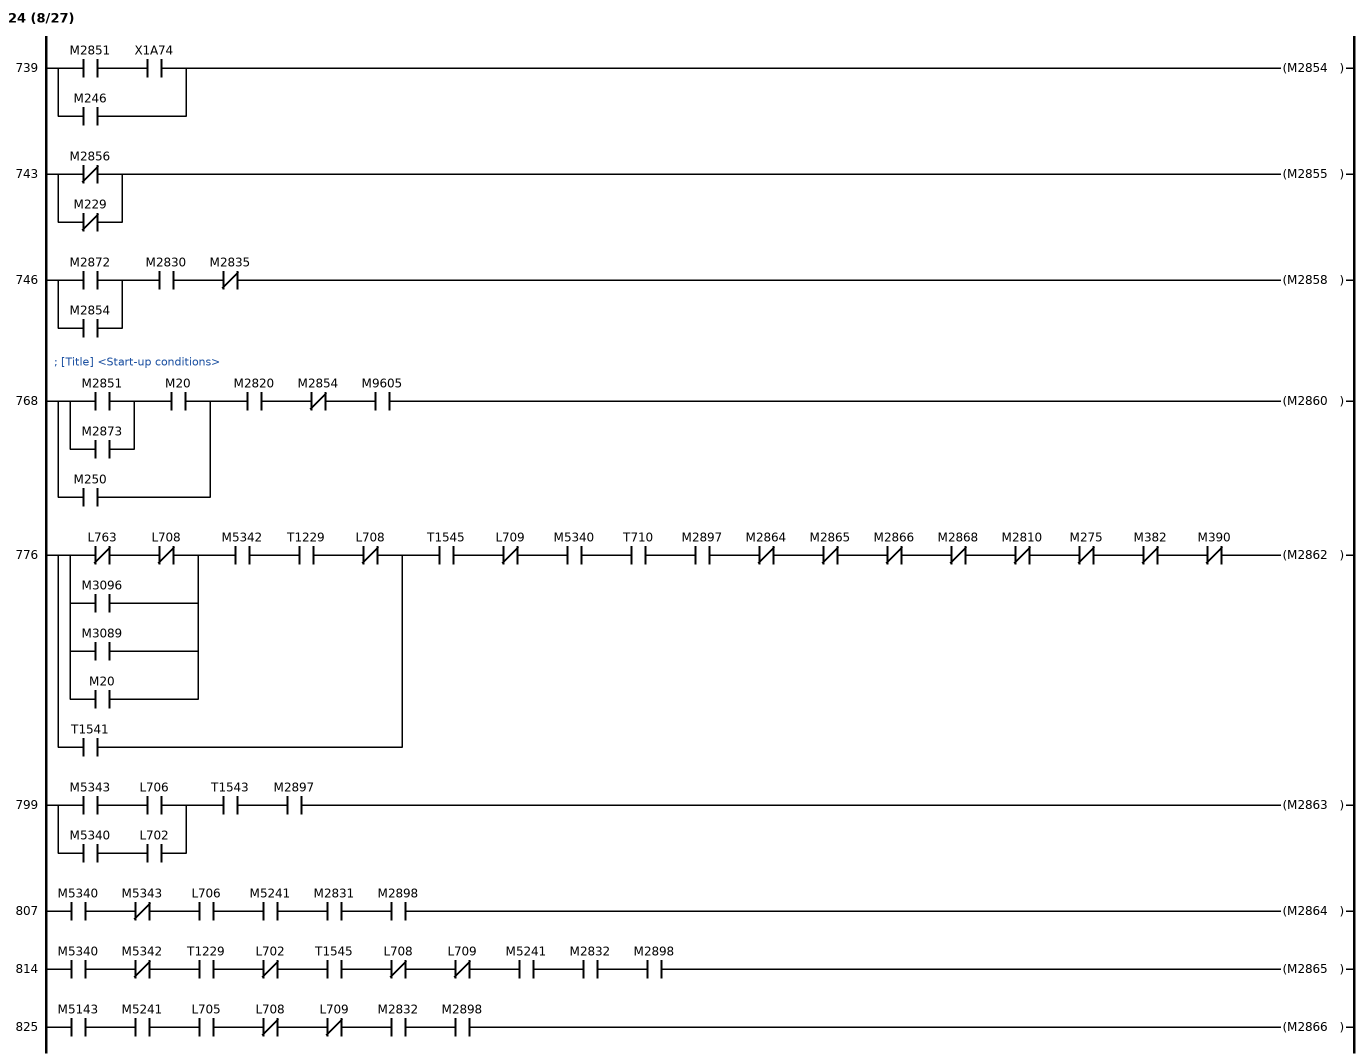
739   LD      M2851
      AND     X1A74
      OR      M246
      OUT     M2854
743   LDI     M2856
      ORI     M229
      OUT     M2855
746   LD      M2872
      OR      M2854
      AND     M2830
      ANI     M2835
      OUT     M2858
; [Title] <Start-up conditions>
768   LD      M2851
      OR      M2873
      AND     M20
      OR      M250
      AND     M2820
      ANI     M2854
      AND     M9605
      OUT     M2860
776   LDI     L763
      ANI     L708
      OR      M3096
      OR      M3089
      OR      M20
      AND     M5342
      AND     T1229
      ANI     L708
      OR      T1541
      AND     T1545
      ANI     L709
      AND     M5340
      AND     T710
      AND     M2897
      ANI     M2864
      ANI     M2865
      ANI     M2866
      ANI     M2868
      ANI     M2810
      ANI     M275
      ANI     M382
      ANI     M390
      OUT     M2862
799   LD      M5343
      AND     L706
      LD      M5340
      AND     L702
      ORB
      AND     T1543
      AND     M2897
      OUT     M2863
807   LD      M5340
      ANI     M5343
      AND     L706
      AND     M5241
      AND     M2831
      AND     M2898
      OUT     M2864
814   LD      M5340
      ANI     M5342
      AND     T1229
      ANI     L702
      AND     T1545
      ANI     L708
      ANI     L709
      AND     M5241
      AND     M2832
      AND     M2898
      OUT     M2865
825   LD      M5143
      AND     M5241
      AND     L705
      ANI     L708
      ANI     L709
      AND     M2832
      AND     M2898
      OUT     M2866
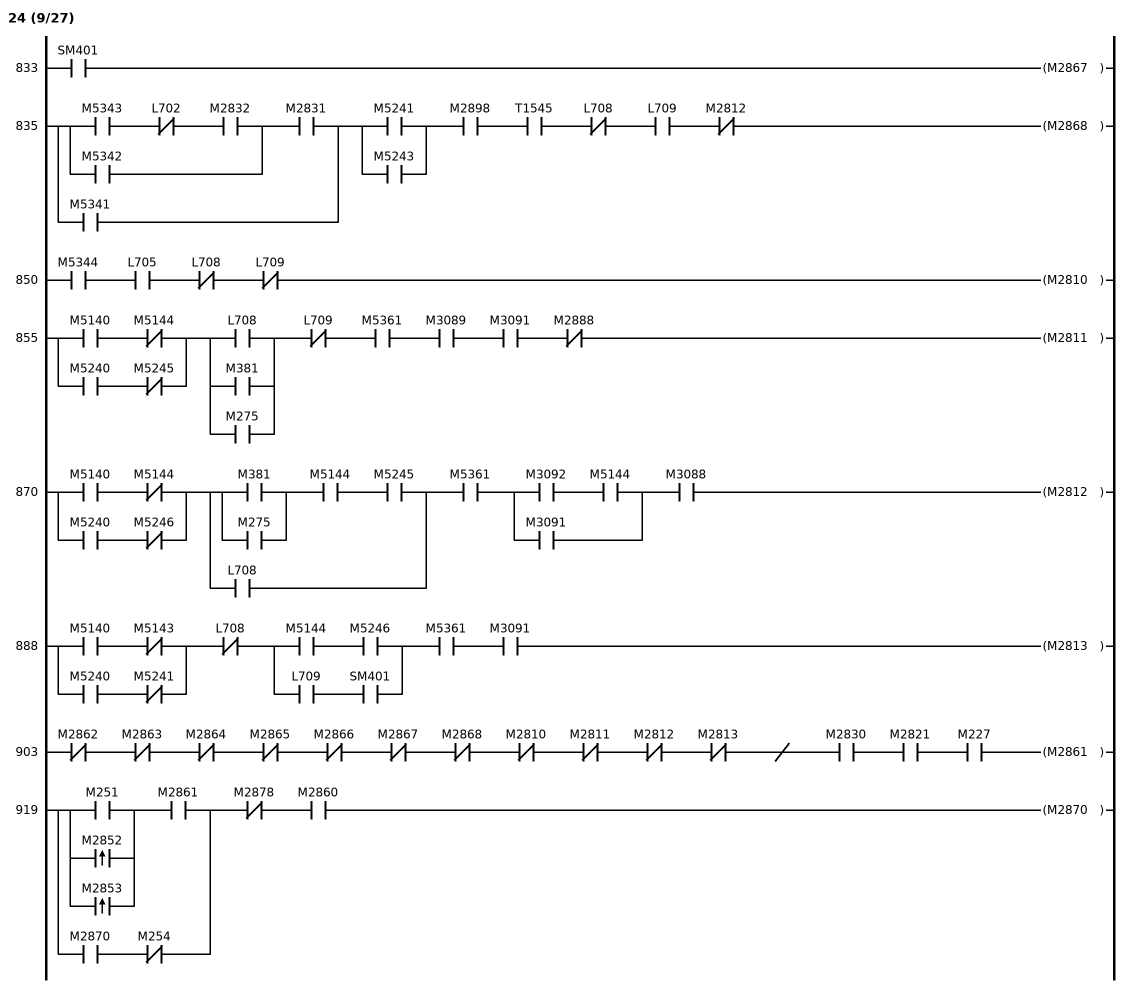
833   LD      SM401
      OUT     M2867
835   LD      M5343
      ANI     L702
      AND     M2832
      OR      M5342
      AND     M2831
      OR      M5341
      LD      M5241
      OR      M5243
      ANB
      AND     M2898
      AND     T1545
      ANI     L708
      AND     L709
      ANI     M2812
      OUT     M2868
850   LD      M5344
      AND     L705
      ANI     L708
      ANI     L709
      OUT     M2810
855   LD      M5140
      ANI     M5144
      LD      M5240
      ANI     M5245
      ORB
      LD      L708
      OR      M381
      OR      M275
      ANB
      ANI     L709
      AND     M5361
      AND     M3089
      AND     M3091
      ANI     M2888
      OUT     M2811
870   LD      M5140
      ANI     M5144
      LD      M5240
      ANI     M5246
      ORB
      LD      M381
      OR      M275
      AND     M5144
      AND     M5245
      OR      L708
      ANB
      AND     M5361
      LD      M3092
      AND     M5144
      OR      M3091
      ANB
      AND     M3088
      OUT     M2812
888   LD      M5140
      ANI     M5143
      LD      M5240
      ANI     M5241
      ORB
      ANI     L708
      LD      M5144
      AND     M5246
      LD      L709
      AND     SM401
      ORB
      ANB
      AND     M5361
      AND     M3091
      OUT     M2813
903   LDI     M2862
      ANI     M2863
      ANI     M2864
      ANI     M2865
      ANI     M2866
      ANI     M2867
      ANI     M2868
      ANI     M2810
      ANI     M2811
      ANI     M2812
      ANI     M2813
      INV
      AND     M2830
      AND     M2821
      AND     M227
      OUT     M2861
919   LD      M251
      ORP     M2852
      ORP     M2853
      AND     M2861
      LD      M2870
      ANI     M254
      ORB
      ANI     M2878
      AND     M2860
      OUT     M2870
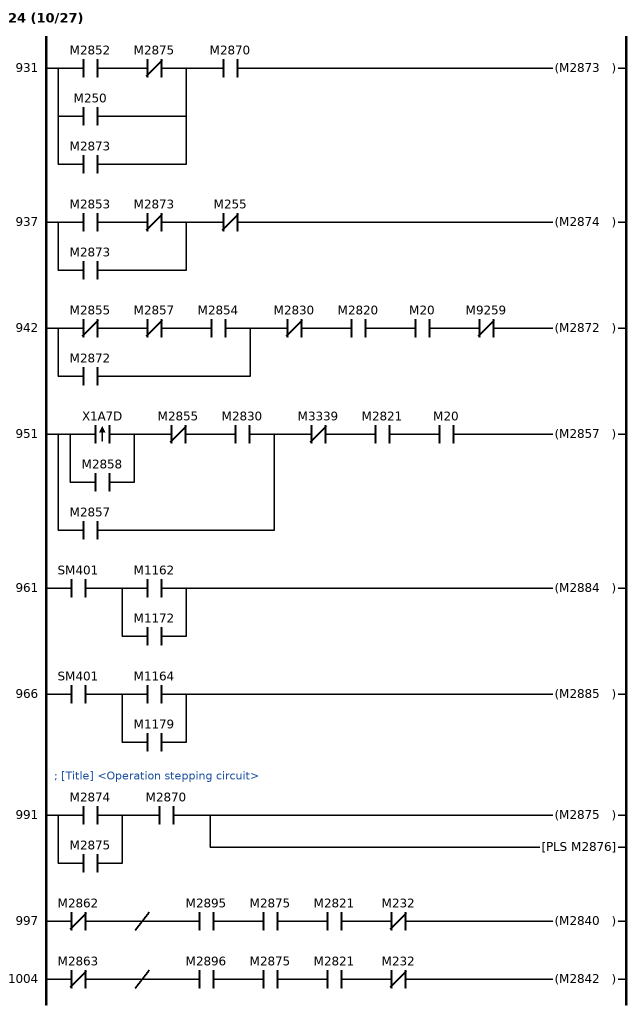
931   LD      M2852
      ANI     M2875
      OR      M250
      OR      M2873
      AND     M2870
      OUT     M2873
937   LD      M2853
      ANI     M2873
      OR      M2873
      ANI     M255
      OUT     M2874
942   LDI     M2855
      ANI     M2857
      AND     M2854
      OR      M2872
      ANI     M2830
      AND     M2820
      AND     M20
      ANI     M9259
      OUT     M2872
951   LDP     X1A7D
      OR      M2858
      ANI     M2855
      AND     M2830
      OR      M2857
      ANI     M3339
      AND     M2821
      AND     M20
      OUT     M2857
961   LD      SM401
      LD      M1162
      OR      M1172
      ANB
      OUT     M2884
966   LD      SM401
      LD      M1164
      OR      M1179
      ANB
      OUT     M2885
; [Title] <Operation stepping circuit>
991   LD      M2874
      OR      M2875
      AND     M2870
      OUT     M2875
      PLS     M2876
997   LDI     M2862
      INV
      AND     M2895
      AND     M2875
      AND     M2821
      ANI     M232
      OUT     M2840
1004  LDI     M2863
      INV
      AND     M2896
      AND     M2875
      AND     M2821
      ANI     M232
      OUT     M2842
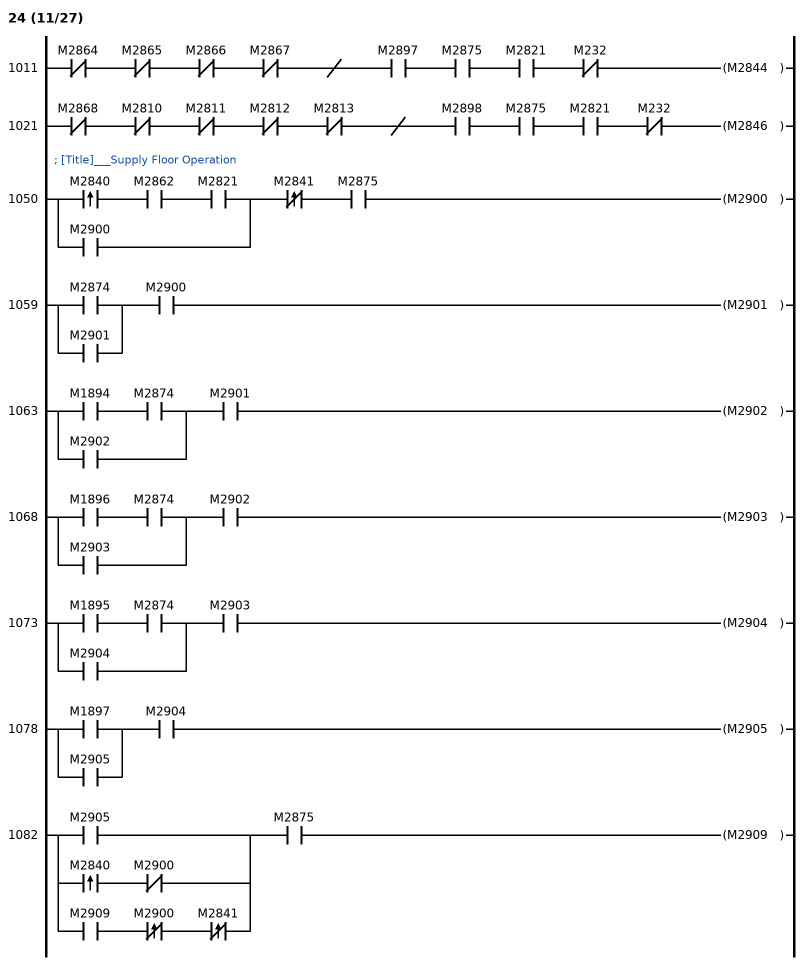
1011  LDI     M2864
      ANI     M2865
      ANI     M2866
      ANI     M2867
      INV
      AND     M2897
      AND     M2875
      AND     M2821
      ANI     M232
      OUT     M2844
1021  LDI     M2868
      ANI     M2810
      ANI     M2811
      ANI     M2812
      ANI     M2813
      INV
      AND     M2898
      AND     M2875
      AND     M2821
      ANI     M232
      OUT     M2846
; [Title]___Supply Floor Operation
1050  LDP     M2840
      AND     M2862
      AND     M2821
      OR      M2900
      ANDPI   M2841
      AND     M2875
      OUT     M2900
1059  LD      M2874
      OR      M2901
      AND     M2900
      OUT     M2901
1063  LD      M1894
      AND     M2874
      OR      M2902
      AND     M2901
      OUT     M2902
1068  LD      M1896
      AND     M2874
      OR      M2903
      AND     M2902
      OUT     M2903
1073  LD      M1895
      AND     M2874
      OR      M2904
      AND     M2903
      OUT     M2904
1078  LD      M1897
      OR      M2905
      AND     M2904
      OUT     M2905
1082  LD      M2905
      LDP     M2840
      ANI     M2900
      ORB
      LD      M2909
      ANDPI   M2900
      ANDPI   M2841
      ORB
      AND     M2875
      OUT     M2909
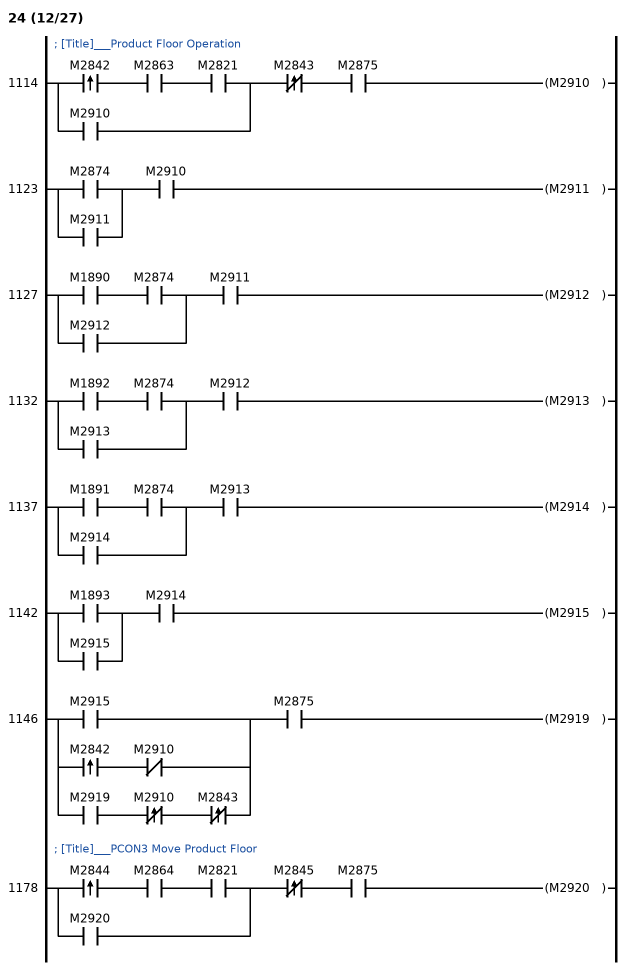
; [Title]___Product Floor Operation
1114  LDP     M2842
      AND     M2863
      AND     M2821
      OR      M2910
      ANDPI   M2843
      AND     M2875
      OUT     M2910
1123  LD      M2874
      OR      M2911
      AND     M2910
      OUT     M2911
1127  LD      M1890
      AND     M2874
      OR      M2912
      AND     M2911
      OUT     M2912
1132  LD      M1892
      AND     M2874
      OR      M2913
      AND     M2912
      OUT     M2913
1137  LD      M1891
      AND     M2874
      OR      M2914
      AND     M2913
      OUT     M2914
1142  LD      M1893
      OR      M2915
      AND     M2914
      OUT     M2915
1146  LD      M2915
      LDP     M2842
      ANI     M2910
      ORB
      LD      M2919
      ANDPI   M2910
      ANDPI   M2843
      ORB
      AND     M2875
      OUT     M2919
; [Title]___PCON3 Move Product Floor
1178  LDP     M2844
      AND     M2864
      AND     M2821
      OR      M2920
      ANDPI   M2845
      AND     M2875
      OUT     M2920
